(* PLC project ARR NG V1.0, SoMachine Motion Logic Builder V1.56.49.0, author SESA100920 *)
(* stored: creationDateTime 2020-05-25T16:35:19.8150034, version 0.0.0.0, modificationDateTime 2020-05-15T14:58:38.6738722 *)

PROGRAM RobotParser
  VAR
    sIp : STRING(15) := '10.139.10.6';
    uiPort : UINT := 5007;
    fbUdpPeer : TCPUDP.FB_UDPPeer;
    stStringToSend : STRING;
    udiSize : UDINT;
    iVal : INT;
    stX : STRING;
    stY : STRING;
    stZ : STRING;
    stRX : STRING;
    stRY : STRING;
    stRZ : STRING;
    stX2 : STRING;
    stY2 : STRING;
    stZ2 : STRING;
    stRX2 : STRING;
    stRY2 : STRING;
    stRZ2 : STRING;
    stNum : STRING;
    stRobot1 : STRING;
    stRObot2 : STRING;
  END_VAR

            CASE iVal OF
	0: IF fbUdpPeer.Open() THEN
		iVal := 1;
		END_IF
		
	1: 	
			stNum := '2';
			stX := CONCAT('X', LREAL_TO_STRING(SR_MainMachine.astExtRobotItf[1].stParam.stRobotData.lrOffsetRobotToMC_X));
			stY := CONCAT('Y', LREAL_TO_STRING(SR_MainMachine.astExtRobotItf[1].stParam.stRobotData.lrOffsetRobotToMC_Y));
			stZ := CONCAT('Z', LREAL_TO_STRING(SR_MainMachine.astExtRobotItf[1].stParam.stRobotData.lrOffset_Z_Robot));
			stRX := CONCAT('RX', LREAL_TO_STRING(SR_MainMachine.astExtRobotItf[1].stParam.stRobotData.lrRotationAngle_Robot_rX));
			stRY := CONCAT('RY', LREAL_TO_STRING(SR_MainMachine.astExtRobotItf[1].stParam.stRobotData.lrRotationAngle_Robot_rY));
			stRZ := CONCAT('RZ', LREAL_TO_STRING(SR_MainMachine.astExtRobotItf[1].stParam.stRobotData.lrRotationAngle_Robot_rZ));
			
			stX2 := CONCAT('X', LREAL_TO_STRING(SR_MainMachine.astExtRobotItf[2].stParam.stRobotData.lrOffsetRobotToMC_X));
			stY2 := CONCAT('Y', LREAL_TO_STRING(SR_MainMachine.astExtRobotItf[2].stParam.stRobotData.lrOffsetRobotToMC_Y));
			stZ2 := CONCAT('Z', LREAL_TO_STRING(SR_MainMachine.astExtRobotItf[2].stParam.stRobotData.lrOffset_Z_Robot));
			stRX2 := CONCAT('RX', LREAL_TO_STRING(SR_MainMachine.astExtRobotItf[2].stParam.stRobotData.lrRotationAngle_Robot_rX));
			stRY2 := CONCAT('RY', LREAL_TO_STRING(SR_MainMachine.astExtRobotItf[2].stParam.stRobotData.lrRotationAngle_Robot_rY));
			stRZ2 := CONCAT('RZ', LREAL_TO_STRING(SR_MainMachine.astExtRobotItf[2].stParam.stRobotData.lrRotationAngle_Robot_rZ));
			
			stRobot1 := CONCAT(stNum, CONCAT(stX, CONCAT(stY, CONCAT(stZ, CONCAT(stRX, CONCAT(stRY, stRZ))))));
			stRobot2 := CONCAT(stX2, CONCAT(stY2, CONCAT(stZ2, CONCAT(stRX2, CONCAT(stRY2, stRZ2)))));
			
			stStringToSend := CONCAT(stRobot1, stRobot2);
			udiSize := SIZEOF(stStringToSend);
			fbUdpPeer.SendTo(sIp, uiPort, ADR(stStringToSend), udiSize);
		
END_CASE
          
END_PROGRAM
